FUNCTION_BLOCK SubSubSystemButtonWidget EXTENDS SubSystemButtonWidget
VAR_INPUT
END_VAR
VAR_IN_OUT
END_VAR
VAR_OUTPUT
END_VAR
VAR
END_VAR

SUPER^(activeTab := activeTab);

END_FUNCTION_BLOCK

(* stored: Version 1.1.0.1, ProductVersion 3.1.4018.2
   POU SubSubSystemButtonWidget: Id {9e9c5463-4f44-4f57-836e-ed90d1a381d9}, SpecialFunc None *)
